(* IEC 61131-3 sources: ST_L/Practice/01_Basic, 4 files *)

(* ---- 01_01_HelloWorld.st ---- *)
(* ============================================================================
 * 文件: 01_01_HelloWorld.st
 * 章节: 第1章 - ST语言简介
 * 描述: 第一个ST程序 - 闪烁灯控制
 * 学习目标: 理解ST程序的基本结构
 * ============================================================================ *)

(* --------------------------------------------------------------------------
 * 全局变量声明
 * 这些变量会被映射到实际的物理输入/输出
 * -------------------------------------------------------------------------- *)
VAR_GLOBAL
    // 数字量输入
    iStartButton AT %IX0.0 : BOOL;      // 启动按钮
    iStopButton AT %IX0.1 : BOOL;      // 停止按钮
    iEmergencyStop AT %IX0.2 : BOOL;    // 急停按钮

    // 数字量输出
    qIndicatorLight AT %QX0.0 : BOOL;   // 指示灯
    qMotorRun AT %QX0.1 : BOOL;         // 电机运行
    qAlarm AT %QX0.2 : BOOL;            // 报警输出

    // 模拟量输入
    iTemperature AT %IW0 : INT;          // 温度传感器
    iPressure AT %IW2 : INT;             // 压力传感器

    // 模拟量输出
    qMotorSpeed AT %QW0 : INT;          // 电机速度设定
END_VAR

(* ============================================================================
 * 程序: HelloWorld
 * 功能: 简单的闪烁灯程序，展示ST程序的基本结构
 * ============================================================================ *)
PROGRAM HelloWorld
VAR
    // 内部变量
    timer : TON;                         // 通电延时定时器
    blinkFlag : BOOL := FALSE;           // 闪烁标志
    cycleCounter : INT := 0;             // 循环计数器
    lastButtonState : BOOL := FALSE;     // 上次按钮状态
    pressCount : INT := 0;               // 按钮按下次数
END_VAR

// ============================================================================
// 主程序逻辑
// ============================================================================
BEGIN
    // ------------------------------------------------------------------------
    // 1. 边沿检测 - 检测启动按钮的上升沿
    // ------------------------------------------------------------------------
    IF iStartButton AND NOT lastButtonState THEN
        pressCount := pressCount + 1;
    END_IF
    lastButtonState := iStartButton;

    // ------------------------------------------------------------------------
    // 2. 急停处理 - 最高优先级
    // ------------------------------------------------------------------------
    IF iEmergencyStop THEN
        qMotorRun := FALSE;
        qAlarm := TRUE;
        blinkFlag := FALSE;
        qIndicatorLight := FALSE;
    ELSE
        qAlarm := FALSE;

        // ------------------------------------------------------------------------
        // 3. 正常启停控制
        // ------------------------------------------------------------------------
        IF iStartButton THEN
            qMotorRun := TRUE;
        END_IF;

        IF iStopButton THEN
            qMotorRun := FALSE;
            blinkFlag := FALSE;
        END_IF;
    END_IF

    // ------------------------------------------------------------------------
    // 4. 闪烁灯逻辑
    // ------------------------------------------------------------------------
    // 当电机运行时，指示灯以1Hz频率闪烁
    timer(IN := NOT timer.Q, PT := T#500ms);

    IF timer.Q THEN
        IF qMotorRun THEN
            blinkFlag := NOT blinkFlag;
        ELSE
            blinkFlag := FALSE;
        END_IF;
    END_IF;

    qIndicatorLight := blinkFlag;

    // ------------------------------------------------------------------------
    // 5. 电机速度控制 - 根据温度调整
    // ------------------------------------------------------------------------
    IF qMotorRun THEN
        // 温度越高，速度越慢（保护电机）
        IF iTemperature < 500 THEN
            qMotorSpeed := 1500;  // 正常速度
        ELSIF iTemperature < 800 THEN
            qMotorSpeed := 1000;  // 中等速度
        ELSE
            qMotorSpeed := 500;   // 低速
        END_IF;
    ELSE
        qMotorSpeed := 0;
    END_IF

    // ------------------------------------------------------------------------
    // 6. 循环计数器
    // ------------------------------------------------------------------------
    cycleCounter := cycleCounter + 1;
    IF cycleCounter >= 1000 THEN
        cycleCounter := 0;
    END_IF;

END_PROGRAM

(* ---- 01_02_VariableDemo.st ---- *)
(* ============================================================================
 * 文件: 01_02_VariableDemo.st
 * 章节: 第2章 - 变量声明与数据类型
 * 描述: 变量声明的完整演示
 * 学习目标: 掌握各种变量的声明方式
 * ============================================================================ *)

PROGRAM VariableDemo
VAR
    // ==========================================================================
    // 1. 基本数据类型声明
    // ==========================================================================

    // 布尔型变量
    bRunning : BOOL := FALSE;           // 带初始值
    bEnabled : BOOL;                    // 默认FALSE
    bFlag : BOOL := 1;                  // 也可用0/1赋值

    // 整数类型
    iCounter : INT := 0;               // 16位整数 -32,768~32,767
    iLargeCounter : DINT := 0;          // 32位整数
    iSmallValue : SINT := -10;         // 8位整数
    iPositive : UINT := 100;            // 无符号整数
    iByte : USINT := 255;               // 字节 0~255

    // 浮点数类型
    fRatio : REAL := 1.5;               // 单精度浮点
    fPi : LREAL := 3.14159265358979;    // 双精度浮点
    fVoltage : REAL := 220.5;           // 电压值
    fSpeed : LREAL := 1500.75;          // 电机转速

    // 时间类型
    tDelay : TIME := T#2s500ms;         // 延时时间
    tCycle : TIME := T#100ms;           // 周期
    tPowerOn : DATE := D#2024-01-01;    // 日期

    // 字符串类型
    sDeviceName : STRING(20) := 'Motor_A';
    sMessage : STRING(50) := 'System Ready';
    sEmpty : STRING(10);

    // 字节/字类型
    byData : BYTE := 16#AB;             // 十六进制
    wData : WORD := 2#1010101010101010; // 二进制
    dwData : DWORD := 16#12345678;       // 双字

    // ==========================================================================
    // 2. 数组声明
    // ==========================================================================

    // 一维数组
    aiTemperatures : ARRAY[1..7] OF INT := [23, 25, 22, 24, 26, 28, 27];
    abFlags : ARRAY[0..7] OF BOOL := [TRUE, FALSE, TRUE, FALSE, TRUE, FALSE, TRUE, FALSE];

    // 多维数组
    amMatrix : ARRAY[1..3, 1..3] OF INT := [1, 2, 3, 4, 5, 6, 7, 8, 9];

    // 字符串数组
    asDayNames : ARRAY[0..6] OF STRING(10) :=
        ['Sunday', 'Monday', 'Tuesday', 'Wednesday', 'Thursday', 'Friday', 'Saturday'];

    // ==========================================================================
    // 3. 临时计算变量
    // ==========================================================================
    iTemp : INT;
    fTemp : REAL;
    bTemp : BOOL;
END_VAR

// ============================================================================
// 主程序逻辑
// ============================================================================
BEGIN
    // -------------------------------------------------------------------------
    // 1. 布尔运算
    // -------------------------------------------------------------------------
    bRunning := TRUE;
    bEnabled := bRunning AND NOT FALSE;     // 结果: TRUE
    bFlag := bRunning OR FALSE;             // 结果: TRUE
    bTemp := NOT bRunning;                  // 结果: FALSE

    // -------------------------------------------------------------------------
    // 2. 算术运算
    // -------------------------------------------------------------------------
    iCounter := 100 + 50;                   // 加法: 150
    iCounter := 100 - 30;                   // 减法: 70
    iCounter := 10 * 5;                     // 乘法: 50
    iCounter := 100 / 3;                    // 整数除法: 33
    iTemp := 100 MOD 3;                     // 取模: 1

    // -------------------------------------------------------------------------
    // 3. 数组访问
    // -------------------------------------------------------------------------
    iTemp := aiTemperatures[1];             // 第一个元素: 23
    iTemp := aiTemperatures[7];             // 最后一个元素: 27

    // 遍历数组计算平均值
    fTemp := 0.0;
    FOR iTemp := 1 TO 7 DO
        fTemp := fTemp + INT_TO_REAL(aiTemperatures[iTemp]);
    END_FOR;
    fTemp := fTemp / 7.0;                   // 平均温度

    // -------------------------------------------------------------------------
    // 4. 多维数组访问
    // -------------------------------------------------------------------------
    iTemp := amMatrix[1, 1];                 // 第一行第一列: 1
    iTemp := amMatrix[2, 2];                 // 第二行第二列: 5
    iTemp := amMatrix[3, 3];                 // 第三行第三列: 9

    // -------------------------------------------------------------------------
    // 5. 位操作
    // -------------------------------------------------------------------------
    byData := 2#10101010;                    // 设置初始值
    byData.0 := TRUE;                        // 设置最低位
    byData.7 := FALSE;                       // 设置最高位
    bTemp := byData.0;                      // 读取最低位

    // -------------------------------------------------------------------------
    // 6. 字符串操作（部分平台支持）
    // -------------------------------------------------------------------------
    sDeviceName := 'Pump_01';
    sMessage := CONCAT(sDeviceName, '_Running');

    // -------------------------------------------------------------------------
    // 7. 类型转换
    // -------------------------------------------------------------------------
    iTemp := 100;
    fTemp := INT_TO_REAL(iTemp);             // INT -> REAL: 100.0
    iTemp := REAL_TO_INT(3.7);               // REAL -> INT: 3 (截断)
    iTemp := ROUND(3.7);                    // 四舍五入: 4

    // -------------------------------------------------------------------------
    // 8. 变量赋值示例
    // -------------------------------------------------------------------------
    iCounter := iCounter + 1;               // 递增
    fRatio := fRatio * 1.1;                 // 乘以1.1

END_PROGRAM

(* ---- 01_03_DataTypeDemo.st ---- *)
(* ============================================================================
 * 文件: 01_03_DataTypeDemo.st
 * 章节: 第2章 - 变量声明与数据类型
 * 描述: 数据类型完整演示
 * 学习目标: 掌握ST语言所有基本数据类型
 * ============================================================================ *)

PROGRAM DataTypeDemo
VAR
    // ==========================================================================
    // 整数类型
    // ==========================================================================
    siValue : SINT;        // 8位有符号: -128 ~ 127
    usiValue : USINT;       // 8位无符号: 0 ~ 255
    iValue : INT;          // 16位有符号: -32768 ~ 32767
    uiValue : UINT;         // 16位无符号: 0 ~ 65535
    diValue : DINT;        // 32位有符号: ~21亿
    udiValue : UDINT;      // 32位无符号: 0 ~ 42亿
    liValue : LINT;        // 64位有符号
    luiValue : LUID;       // 64位无符号

    // ==========================================================================
    // 浮点数类型
    // ==========================================================================
    rSingle : REAL;        // 32位浮点
    lrDouble : LREAL;      // 64位浮点

    // ==========================================================================
    // 时间日期类型
    // ==========================================================================
    tDuration : TIME;          // 时间段
    dDate : DATE;              // 日期
    todTime : TIME_OF_DAY;     // 一天中的时间
    dtDateTime : DATE_AND_TIME; // 日期时间

    // ==========================================================================
    // 字符串类型
    // ==========================================================================
    sShort : STRING(10);
    sMedium : STRING(50);
    sLong : STRING(255);
    wsWide : WSTRING(100);     // 宽字符串

    // ==========================================================================
    // 位数据
    // ==========================================================================
    byByte : BYTE;         // 8位
    wWord : WORD;          // 16位
    dwDword : DWORD;       // 32位
    lwLword : LWORD;       // 64位

    // ==========================================================================
    // 布尔类型
    // ==========================================================================
    bTrue : BOOL := TRUE;
    bFalse : BOOL := FALSE;
    bOneZero : BOOL := 1;

    // ==========================================================================
    // 临时变量
    // ==========================================================================
    i : INT;
    rTemp : REAL;
    tTemp : TIME;
END_VAR

// ============================================================================
// 主程序逻辑
// ============================================================================
BEGIN
    // ==========================================================================
    // 1. 整数类型赋值
    // ==========================================================================
    siValue := 100;
    usiValue := 200;
    iValue := 30000;
    uiValue := 60000;
    diValue := 2000000000;
    udiValue := 4000000000;

    // 十六进制表示
    byByte := 16#FF;
    wWord := 16#ABCD;
    dwDword := 16#12345678;

    // 二进制表示
    byByte := 2#11110000;
    wWord := 2#1010101010101010;

    // ==========================================================================
    // 2. 浮点数赋值
    // ==========================================================================
    rSingle := 3.14159;
    lrDouble := 3.14159265358979323846;

    // 指数表示
    rSingle := 1.5E+10;     // 15000000000
    rSingle := 1.0E-6;      // 0.000001
    lrDouble := 2.0E+308;   // 非常大的数

    // ==========================================================================
    // 3. 时间类型赋值
    // ==========================================================================
    // 各种时间格式
    tDuration := T#1s;              // 1秒
    tDuration := T#500ms;          // 500毫秒
    tDuration := T#1m30s;          // 1分30秒
    tDuration := T#2h15m30s500ms;  // 2小时15分30秒500毫秒
    tDuration := tDuration + tDuration;  // 时间相加

    // 日期赋值
    dDate := D#2024-01-15;
    todTime := TOD#12:30:45.123;
    dtDateTime := DT#2024-01-15-12:30:45;

    // ==========================================================================
    // 4. 字符串赋值
    // ==========================================================================
    sShort := 'Hi';
    sMedium := 'This is a medium length string';
    sLong := 'This is a very long string that can hold up to 255 characters';

    // ==========================================================================
    // 5. 位访问
    // ==========================================================================
    byByte := 16#00;                   // 清除
    byByte.0 := TRUE;                  // 设置位0
    byByte.7 := TRUE;                  // 设置位7
    bTrue := byByte.0;                 // 读取位0

    wWord := 16#0000;
    wWord.0 := TRUE;                   // 位0
    wWord.15 := TRUE;                  // 位15 (最高位)

    // ==========================================================================
    // 6. 位操作
    // ==========================================================================
    byByte := 2#10101010;

    // 位与
    wWord := 16#F0F0 AND 16#0F0F;     // 结果: 16#0000

    // 位或
    wWord := 16#F0F0 OR 16#0F0F;      // 结果: 16#FFFF

    // 位异或
    wWord := 16#F0F0 XOR 16#FFFF;     // 结果: 16#0F0F

    // 位取反
    byByte := NOT 2#10101010;         // 结果: 2#01010101

    // 移位
    wWord := 2#0001 SHL 4;            // 左移4位: 2#00010000 = 16
    wWord := 2#10000 SHR 4;          // 右移4位: 2#0001 = 1

    // ==========================================================================
    // 7. 类型转换示例
    // ==========================================================================
    // INT -> REAL
    rTemp := INT_TO_REAL(100);        // 100.0

    // REAL -> INT (截断)
    iValue := REAL_TO_INT(3.9);      // 3

    // INT -> WORD (按位解释)
    wWord := INT_TO_WORD(256);       // 16#0100

    // WORD -> INT
    iValue := WORD_TO_INT(16#0100);  // 256

    // BOOL -> INT
    iValue := BOOL_TO_INT(TRUE);     // 1
    iValue := BOOL_TO_INT(FALSE);    // 0

    // INT -> BOOL (非零为TRUE)
    bTrue := INT_TO_BOOL(100);       // TRUE
    bFalse := INT_TO_BOOL(0);       // FALSE

    // ==========================================================================
    // 8. 数值范围展示
    // ==========================================================================
    siValue := 127;                   // SINT最大值
    siValue := -128;                  // SINT最小值
    usiValue := 255;                  // USINT最大值
    iValue := 32767;                  // INT最大值
    iValue := -32768;                 // INT最小值
    uiValue := 65535;                 // UINT最大值

END_PROGRAM

(* ---- 01_04_OperatorDemo.st ---- *)
(* ============================================================================
 * 文件: 01_04_OperatorDemo.st
 * 章节: 第3章 - 运算符与表达式
 * 描述: 运算符完整演示
 * 学习目标: 掌握ST语言所有运算符
 * ============================================================================ *)

PROGRAM OperatorDemo
VAR
    // ==========================================================================
    // 算术运算符演示
    // ==========================================================================
    iA, iB, iResult : INT;
    rX, rY, rResult : REAL;
    diLarge : DINT;

    // ==========================================================================
    // 比较运算符演示
    // ==========================================================================
    bCompare1, bCompare2, bCompare3 : BOOL;
    iValue : INT := 50;

    // ==========================================================================
    // 逻辑运算符演示
    // ==========================================================================
    bLogic1, bLogic2, bLogic3 : BOOL;
    bEnable, bRunning, bAlarm : BOOL;

    // ==========================================================================
    // 位运算符演示
    // ==========================================================================
    byData1, byData2, byResult : BYTE;
    wData, wMask : WORD;

    // ==========================================================================
    // 临时变量
    // ==========================================================================
    i : INT;
END_VAR

// ============================================================================
// 主程序逻辑
// ============================================================================
BEGIN
    // ==========================================================================
    // 1. 算术运算符
    // ==========================================================================
    iA := 20;
    iB := 6;

    // 加法
    iResult := iA + iB;               // 26

    // 减法
    iResult := iA - iB;               // 14

    // 乘法
    iResult := iA * iB;               // 120

    // 整数除法（截断小数）
    iResult := iA / iB;               // 3 (20 / 6 = 3.33...)

    // 取模（余数）
    iResult := iA MOD iB;            // 2 (20 % 6 = 2)

    // 幂运算
    iResult := 2 ** 10;               // 1024
    iResult := 3 ** 4;                // 81

    // ==========================================================================
    // 2. 浮点算术运算
    // ==========================================================================
    rX := 10.0;
    rY := 3.0;

    rResult := rX / rY;               // 3.3333...

    // 负数
    rResult := -rX;                   // -10.0

    // 复合运算
    rResult := (rX + rY) * (rX - rY); // (10+3) * (10-3) = 91

    // ==========================================================================
    // 3. 比较运算符
    // ==========================================================================
    iA := 10;
    iB := 20;

    // 等于
    bCompare1 := (iA = iB);           // FALSE

    // 不等于
    bCompare2 := (iA <> iB);          // TRUE

    // 小于
    bCompare3 := (iA < iB);           // TRUE

    // 大于
    bCompare1 := (iA > iB);           // FALSE

    // 小于等于
    bCompare2 := (iA <= iB);          // TRUE

    // 大于等于
    bCompare3 := (iA >= iB);          // FALSE

    // ==========================================================================
    // 4. 逻辑运算符
    // ==========================================================================
    bEnable := TRUE;
    bRunning := TRUE;
    bAlarm := FALSE;

    // 逻辑与 AND
    bLogic1 := bEnable AND bRunning;   // TRUE AND TRUE = TRUE
    bLogic1 := bEnable AND bAlarm;     // TRUE AND FALSE = FALSE

    // 逻辑或 OR
    bLogic2 := bAlarm OR bRunning;     // FALSE OR TRUE = TRUE
    bLogic2 := bAlarm OR NOT bRunning; // FALSE OR FALSE = FALSE

    // 逻辑异或 XOR
    bLogic3 := bEnable XOR bRunning;   // TRUE XOR TRUE = FALSE
    bLogic3 := bEnable XOR bAlarm;     // TRUE XOR FALSE = TRUE

    // 逻辑非 NOT
    bLogic1 := NOT bAlarm;             // NOT FALSE = TRUE
    bLogic1 := NOT bEnable;            // NOT TRUE = FALSE

    // 复杂逻辑表达式
    bLogic1 := (bEnable AND bRunning) OR bAlarm;          // TRUE
    bLogic1 := bEnable AND (bRunning OR bAlarm);           // TRUE
    bLogic1 := NOT bAlarm AND (bEnable OR bRunning);      // TRUE

    // ==========================================================================
    // 5. 位运算符
    // ==========================================================================
    byData1 := 2#10101010;    // 170
    byData2 := 2#11001100;    // 204

    // 位与
    byResult := byData1 AND byData2;
    // 10101010
    // 11001100
    // --------
    // 10001000 = 136

    // 位或
    byResult := byData1 OR byData2;
    // 10101010
    // 11001100
    // --------
    // 11101110 = 238

    // 位异或
    byResult := byData1 XOR byData2;
    // 10101010
    // 11001100
    // --------
    // 01100110 = 102

    // 位取反
    byResult := NOT byData1;
    // NOT 10101010 = 01010101 = 85

    // ==========================================================================
    // 6. 移位运算符
    // ==========================================================================
    byData1 := 2#00000001;    // 1

    // 左移
    byResult := byData1 SHL 1;    // 2  (00000010)
    byResult := byData1 SHL 2;    // 4  (00000100)
    byResult := byData1 SHL 4;    // 16 (00010000)
    byResult := byData1 SHL 7;    // 128 (10000000)

    // 右移
    byData1 := 2#10000000;    // 128
    byResult := byData1 SHR 1;    // 64 (01000000)
    byResult := byData1 SHR 2;    // 32 (00100000)
    byResult := byData1 SHR 4;    // 8  (00001000)

    // ==========================================================================
    // 7. 复合表达式
    // ==========================================================================
    iA := 10;
    iB := 20;
    rX := 2.5;

    // 运算优先级: NOT > AND > OR
    // 1 + 2 * 3 - 4 / 2
    iResult := 1 + 2 * 3 - 4 / 2;     // 1 + 6 - 2 = 5

    // 使用括号明确优先级
    iResult := ((1 + 2) * (3 - 4)) / 2;   // (3 * -1) / 2 = -1

    // 混合类型
    rResult := INT_TO_REAL(iA) / INT_TO_REAL(iB) * rX;
    // 10.0 / 20.0 * 2.5 = 1.25

    // ==========================================================================
    // 8. 实用计算示例
    // ==========================================================================

    // 计算圆的面积
    rX := 5.0;                         // 半径
    rResult := 3.14159 * rX * rX;     // 面积 = πr²

    // 计算两点距离
    rX := 3.0;   // x1
    rY := 4.0;   // y1
    // 假设 x2=0, y2=0
    rResult := SQRT(rX * rX + rY * rY);  // 距离 = 5

    // 摄氏度转华氏度
    rX := 25.0;                               // 25°C
    rResult := rX * 9.0 / 5.0 + 32.0;       // 77°F

    // 位掩码操作
    wData := 16#ABCD;
    wMask := 16#00FF;

    // 提取低字节
    byResult := LOW_BYTE(wData AND wMask);    // 16#CD

    // 提取高字节
    wMask := 16#FF00;
    byResult := HIGH_BYTE((wData AND wMask) SHR 8);  // 16#AB

END_PROGRAM
